TYPE TcoInsightResultData_v_5_x_x :
STRUCT
    InspectionID AT %I* : UINT;
    ResultCode AT %I* : UINT;
    InspectionResults AT %I* : ARRAY[0..245] OF BYTE;
END_STRUCT
END_TYPE

(* stored: Version 1.1.0.1, ProductVersion 3.1.4024.11
   DUT TcoInsightResultData_v_5_x_x: Id {b20a7b56-12b0-0923-1949-76b167f6baca} *)
